Staubli VAL3: onSave.pgx

public program onSave(string& x_sItem[])
  local num i
  local num l_nSize
begin
  //if bToSave
  // update
  if isDefined(pt:tTraj[pEditPoint.sID])
    pt:tTraj[pEditPoint.sID]=pEditPoint
    call pt:link_all(pEditPoint.sID)
  endIf
  // saveIt
  pt:libSave()
  bToSave=false
  //$fileClose(nFile)
  // endIf
end
